// Mitsubishi GX Works2 project: 산업기사_기출_1   PLC: Q02/Q02H

PROGRAM MAIN
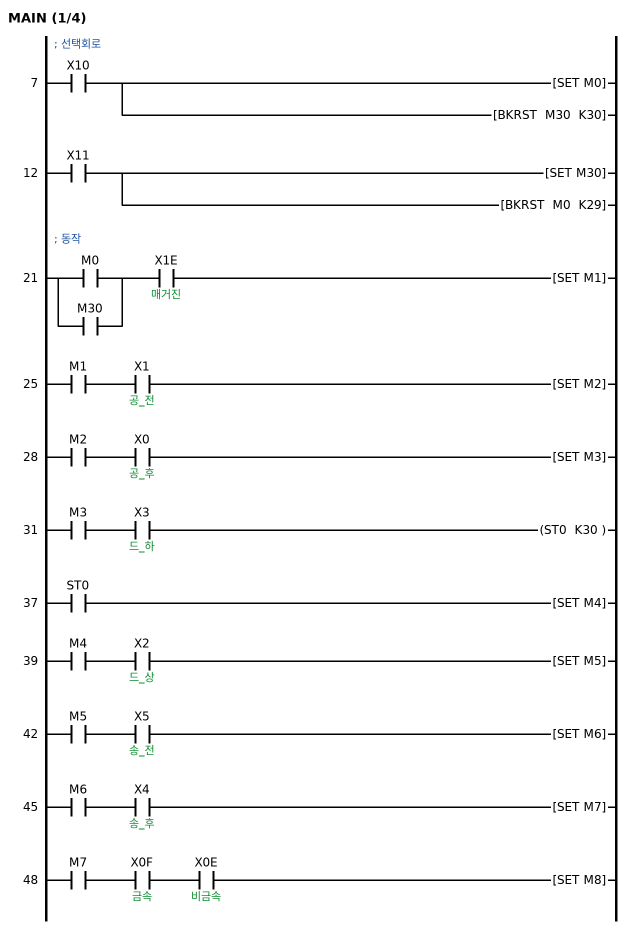
; 선택회로
7     LD      X10
      SET     M0
      BKRST   M30 K30
12    LD      X11
      SET     M30
      BKRST   M0 K29
; 동작
21    LD      M0
      OR      M30
      AND     X1E  ; 매거진
      SET     M1
25    LD      M1
      AND     X1  ; 공_전
      SET     M2
28    LD      M2
      AND     X0  ; 공_후
      SET     M3
31    LD      M3
      AND     X3  ; 드_하
      OUT     ST0 K30
37    LD      ST0
      SET     M4
39    LD      M4
      AND     X2  ; 드_상
      SET     M5
42    LD      M5
      AND     X5  ; 송_전
      SET     M6
45    LD      M6
      AND     X4  ; 송_후
      SET     M7
48    LD      M7
      AND     X0F  ; 금속
      AND     X0E  ; 비금속
      SET     M8
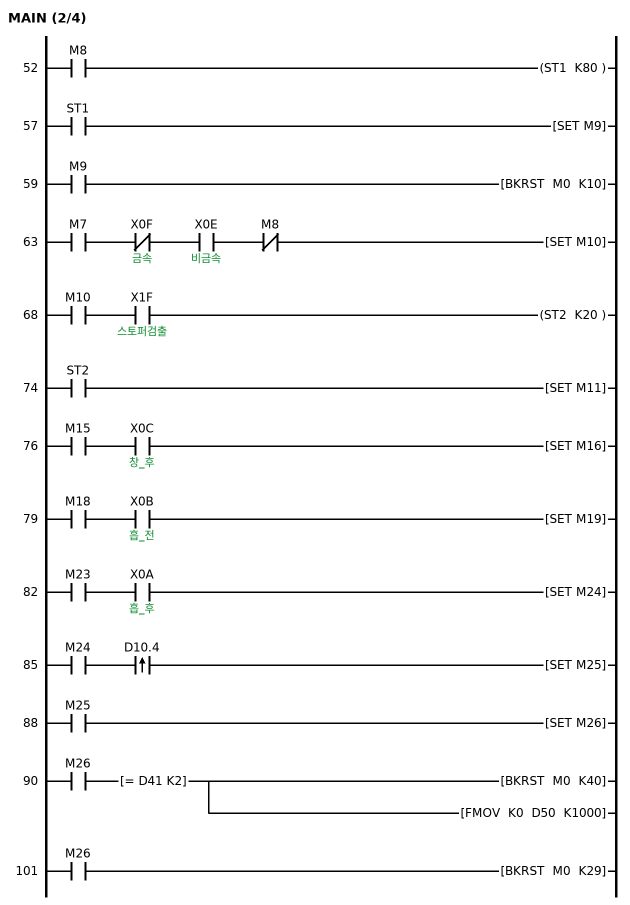
52    LD      M8
      OUT     ST1 K80
57    LD      ST1
      SET     M9
59    LD      M9
      BKRST   M0 K10
63    LD      M7
      ANI     X0F  ; 금속
      AND     X0E  ; 비금속
      ANI     M8
      SET     M10
68    LD      M10
      AND     X1F  ; 스토퍼검출
      OUT     ST2 K20
74    LD      ST2
      SET     M11
76    LD      M15
      AND     X0C  ; 창_후
      SET     M16
79    LD      M18
      AND     X0B  ; 흡_전
      SET     M19
82    LD      M23
      AND     X0A  ; 흡_후
      SET     M24
85    LD      M24
      ANDP    D10.4
      SET     M25
88    LD      M25
      SET     M26
90    LD      M26
      AND=    D41 K2
      BKRST   M0 K40
      FMOV    K0 D50 K1000
101   LD      M26
      BKRST   M0 K29
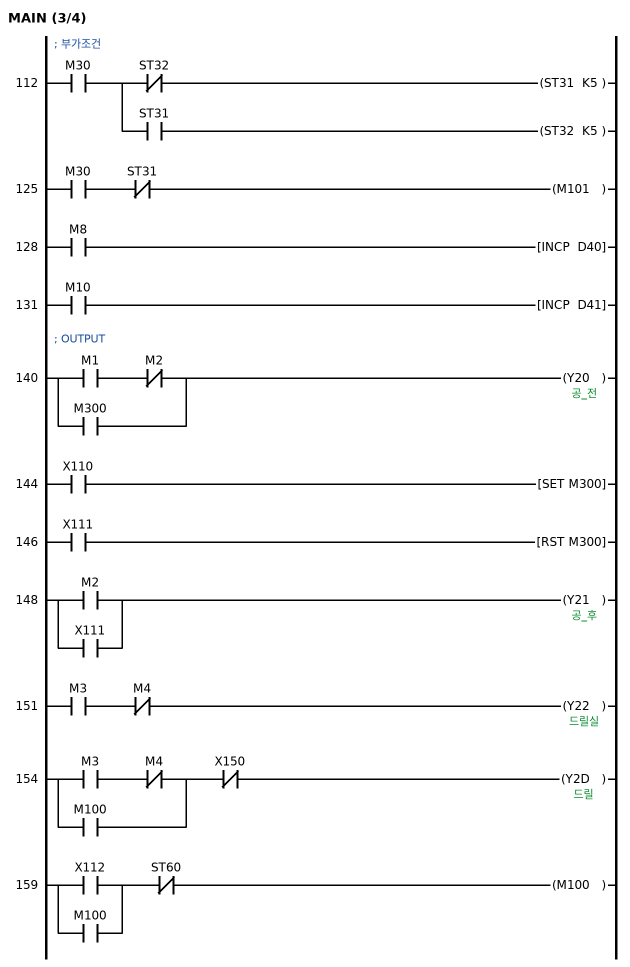
; 부가조건
112   LD      M30
      MPS
      ANI     ST32
      OUT     ST31 K5
      MPP
      AND     ST31
      OUT     ST32 K5
125   LD      M30
      ANI     ST31
      OUT     M101
128   LD      M8
      INCP    D40
131   LD      M10
      INCP    D41
; OUTPUT
140   LD      M1
      ANI     M2
      OR      M300
      OUT     Y20  ; 공_전
144   LD      X110
      SET     M300
146   LD      X111
      RST     M300
148   LD      M2
      OR      X111
      OUT     Y21  ; 공_후
151   LD      M3
      ANI     M4
      OUT     Y22  ; 드릴실
154   LD      M3
      ANI     M4
      OR      M100
      ANI     X150
      OUT     Y2D  ; 드릴
159   LD      X112
      OR      M100
      ANI     ST60
      OUT     M100
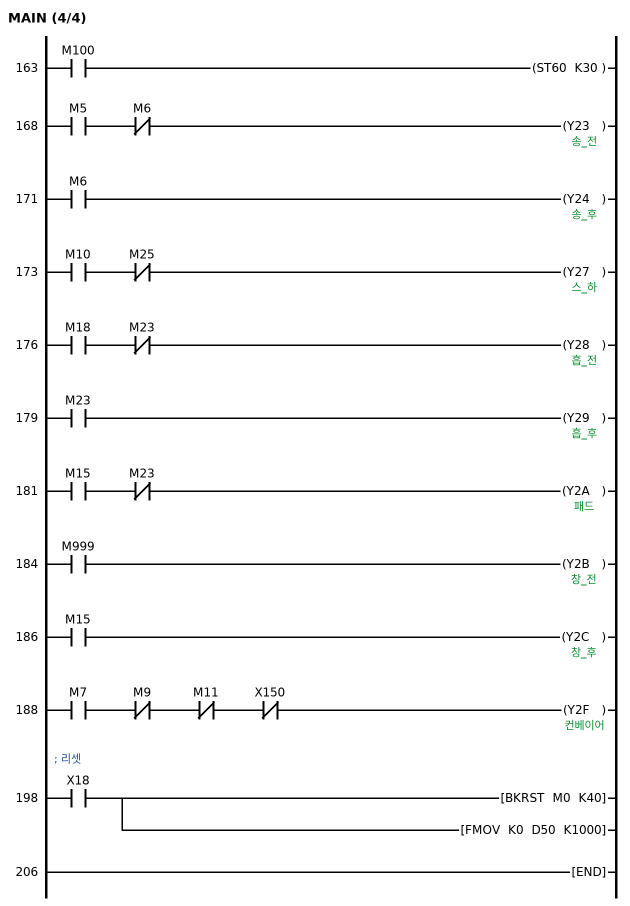
163   LD      M100
      OUT     ST60 K30
168   LD      M5
      ANI     M6
      OUT     Y23  ; 송_전
171   LD      M6
      OUT     Y24  ; 송_후
173   LD      M10
      ANI     M25
      OUT     Y27  ; 스_하
176   LD      M18
      ANI     M23
      OUT     Y28  ; 흡_전
179   LD      M23
      OUT     Y29  ; 흡_후
181   LD      M15
      ANI     M23
      OUT     Y2A  ; 패드
184   LD      M999
      OUT     Y2B  ; 창_전
186   LD      M15
      OUT     Y2C  ; 창_후
188   LD      M7
      ANI     M9
      ANI     M11
      ANI     X150
      OUT     Y2F  ; 컨베이어
; 리셋
198   LD      X18
      BKRST   M0 K40
      FMOV    K0 D50 K1000
206   END
END_PROGRAM

PROGRAM SERVO
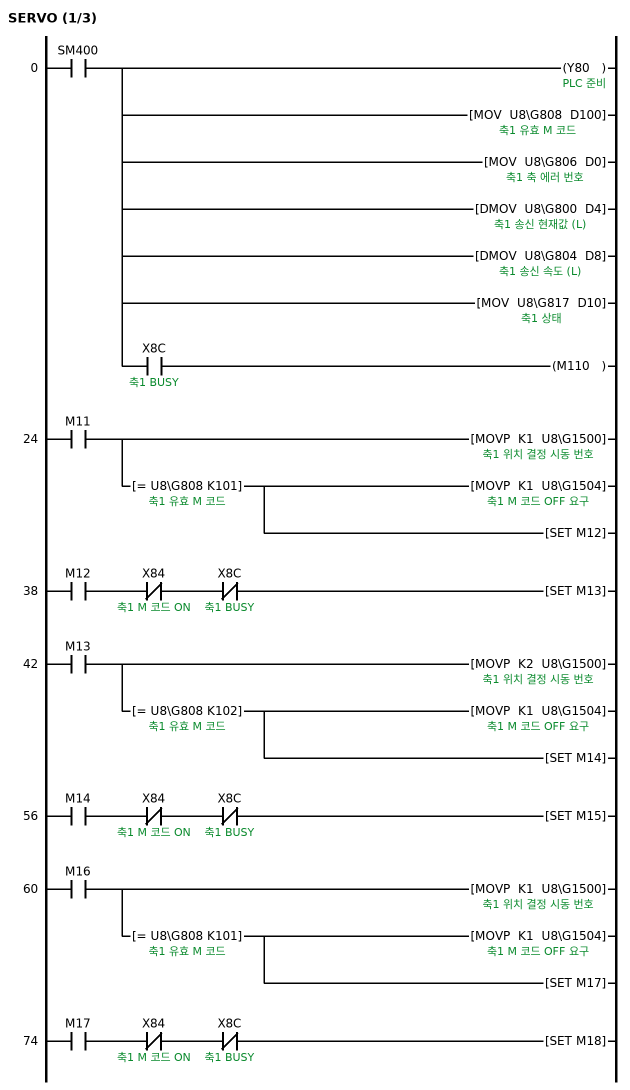
0     LD      SM400
      OUT     Y80  ; PLC 준비
      MOV     U8\G808 D100  ; 축1 유효 M 코드
      MOV     U8\G806 D0  ; 축1 축 에러 번호
      DMOV    U8\G800 D4  ; 축1 송신 현재값 (L)
      DMOV    U8\G804 D8  ; 축1 송신 속도 (L)
      MOV     U8\G817 D10  ; 축1 상태
      AND     X8C  ; 축1 BUSY
      OUT     M110
24    LD      M11
      MOVP    K1 U8\G1500  ; 축1 위치 결정 시동 번호
      AND=    U8\G808 K101  ; 축1 유효 M 코드
      MOVP    K1 U8\G1504  ; 축1 M 코드 OFF 요구
      SET     M12
38    LD      M12
      ANI     X84  ; 축1 M 코드 ON
      ANI     X8C  ; 축1 BUSY
      SET     M13
42    LD      M13
      MOVP    K2 U8\G1500
      AND=    U8\G808 K102  ; 축1 유효 M 코드
      MOVP    K1 U8\G1504
      SET     M14
56    LD      M14
      ANI     X84  ; 축1 M 코드 ON
      ANI     X8C  ; 축1 BUSY
      SET     M15
60    LD      M16
      MOVP    K1 U8\G1500
      AND=    U8\G808 K101  ; 축1 유효 M 코드
      MOVP    K1 U8\G1504
      SET     M17
74    LD      M17
      ANI     X84  ; 축1 M 코드 ON
      ANI     X8C  ; 축1 BUSY
      SET     M18
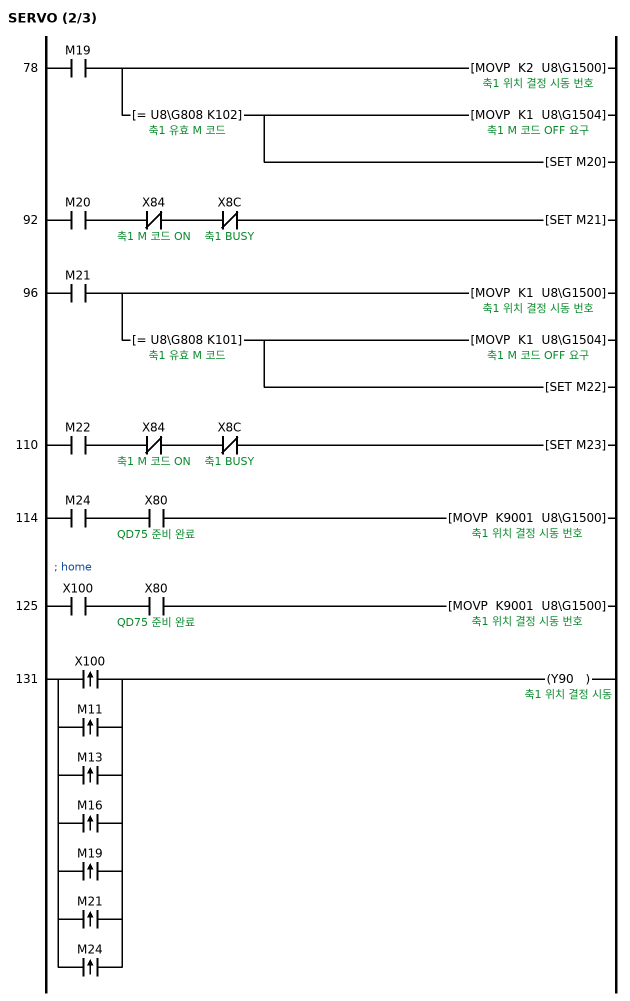
78    LD      M19
      MOVP    K2 U8\G1500
      AND=    U8\G808 K102  ; 축1 유효 M 코드
      MOVP    K1 U8\G1504
      SET     M20
92    LD      M20
      ANI     X84  ; 축1 M 코드 ON
      ANI     X8C  ; 축1 BUSY
      SET     M21
96    LD      M21
      MOVP    K1 U8\G1500
      AND=    U8\G808 K101  ; 축1 유효 M 코드
      MOVP    K1 U8\G1504
      SET     M22
110   LD      M22
      ANI     X84  ; 축1 M 코드 ON
      ANI     X8C  ; 축1 BUSY
      SET     M23
114   LD      M24
      AND     X80  ; QD75 준비 완료
      MOVP    K9001 U8\G1500
; home
125   LD      X100
      AND     X80  ; QD75 준비 완료
      MOVP    K9001 U8\G1500
131   LDP     X100
      ORP     M11
      ORP     M13
      ORP     M16
      ORP     M19
      ORP     M21
      ORP     M24
      OUT     Y90  ; 축1 위치 결정 시동
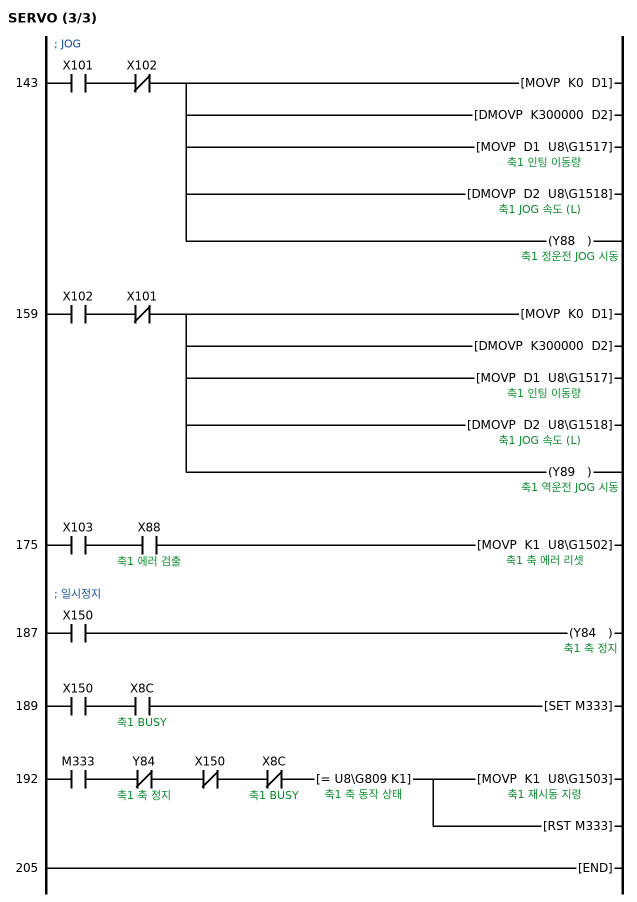
; JOG
143   LD      X101
      ANI     X102
      MOVP    K0 D1
      DMOVP   K300000 D2
      MOVP    D1 U8\G1517  ; 축1 인팅 이동량
      DMOVP   D2 U8\G1518  ; 축1 JOG 속도 (L)
      OUT     Y88  ; 축1 정운전 JOG 시동
159   LD      X102
      ANI     X101
      MOVP    K0 D1
      DMOVP   K300000 D2
      MOVP    D1 U8\G1517
      DMOVP   D2 U8\G1518
      OUT     Y89  ; 축1 역운전 JOG 시동
175   LD      X103
      AND     X88  ; 축1 에러 검출
      MOVP    K1 U8\G1502  ; 축1 축 에러 리셋
; 일시정지
187   LD      X150
      OUT     Y84  ; 축1 축 정지
189   LD      X150
      AND     X8C  ; 축1 BUSY
      SET     M333
192   LD      M333
      ANI     Y84  ; 축1 축 정지
      ANI     X150
      ANI     X8C  ; 축1 BUSY
      AND=    U8\G809 K1  ; 축1 축 동작 상태
      MOVP    K1 U8\G1503  ; 축1 재시동 지령
      RST     M333
205   END
END_PROGRAM

// device comments not shown above
X6  ; 배_후
X7  ; 배_전
X8  ; 스_상
X9  ; 스_하
X0D  ; 창_전
X81  ; 동기용 플래그
X85  ; 축2 M 코드 ON
X89  ; 축2 에러 검출
X8D  ; 축2 BUSY
X90  ; 축1 시동 완료
X91  ; 축2 시동 완료
X94  ; 축1 위치 결정 완료
X95  ; 축2 위치 결정 완료
Y25  ; 배_전
Y26  ; 배_후
Y85  ; 축2 축 정지
Y8A  ; 축2 정운전 JOG 시동
Y8B  ; 축2 역운전 JOG 시동
Y91  ; 축2 위치 결정 시동
Y94  ; 축1 실행 금지 플래그
Y95  ; 축2 실행 금지 플래그
